% RSLogix 500 project LVD211007_994.RSS, saved by version 12.00.00.00 %
PROJECT "LINL0619"    % processor: MicroLogix 1400 %

PROGRAM FILES
  LAD 2 "MAIN"  70 rungs  % Main Program Routine %
  LAD 3 "FAST_TRIG"  9 rungs
  LAD 4 "ENABLES"  19 rungs
  LAD 5 "FEED"  14 rungs  % normal %
  LAD 6 "SPEEDS"  22 rungs
  LAD 7 "HSC BOT"  5 rungs
  LAD 8 "HSC TOP"  5 rungs
  LAD 9 "1 MS STI"  25 rungs  % high speed %
  LAD 10 "SHIFT BOT"  5 rungs
  LAD 11 "SHIFT TOP"  6 rungs
  LAD 12 "BOTOPTIC"  3 rungs
  LAD 13 "BOTOPTMES"  7 rungs
  LAD 14 "SHIFT TOP2"  7 rungs  % shift top inspection 6 %
  LAD 81 "I1"  25 rungs
  LAD 82 "I1 RESULT"  12 rungs
  LAD 83 "I1 PASS"  3 rungs
  LAD 84 "I1 FAIL"  3 rungs
  LAD 85 "I1 ACQ"  9 rungs
  LAD 86 "I1 TESTER"  5 rungs
  LAD 87 "I1 TRIG"  5 rungs
  LAD 88 "NO FIFO"  1 rungs
  LAD 89 "NO FIFO"  1 rungs
  LAD 90 "I1 DATA"  3 rungs
  LAD 91 "I1 FAULT"  9 rungs
  LAD 92 "I1 FIX1"  5 rungs
  LAD 93 "I1 FIX2"  3 rungs
  LAD 94 "I2"  24 rungs
  LAD 95 "I2 RESULT"  11 rungs
  LAD 96 "I2 PASS"  3 rungs
  LAD 97 "I2 FAIL"  3 rungs
  LAD 98 "I2 ACQ"  8 rungs
  LAD 99 "I2 TESTER"  9 rungs
  LAD 100 "I2 TRIG"  5 rungs
  LAD 101 "I2 FIFOSET"  7 rungs
  LAD 102 "I2 FIFOGET"  8 rungs
  LAD 103 "I2 DATA"  3 rungs
  LAD 104 "I2 FAULT"  9 rungs
  LAD 105 "I2 FIX1"  7 rungs
  LAD 106 "I2 FIX2"  3 rungs
  LAD 107 "I3"  1 rungs
  LAD 108 "I3 RESULT"  1 rungs
  LAD 109 "I3 PASS"  1 rungs
  LAD 110 "I3 FAIL"  1 rungs
  LAD 111 "I3 ACQ"  1 rungs
  LAD 112 "I3 TESTER"  1 rungs
  LAD 113 "I3 TRIG"  1 rungs
  LAD 114 "I3 FIFOSET"  1 rungs
  LAD 115 "I3 FIFOGET"  1 rungs
  LAD 116 "I3 DATA"  1 rungs
  LAD 117 "I3 FAULT"  1 rungs
  LAD 118 "I3 FIX1"  1 rungs
  LAD 119 "I3 FIX2"  1 rungs
  LAD 120 "I4"  1 rungs
  LAD 121 "I4 RESULT"  1 rungs
  LAD 122 "I4 PASS"  1 rungs
  LAD 123 "I4 FAIL"  1 rungs
  LAD 124 "I4 ACQ"  1 rungs
  LAD 125 "I4 TESTER"  1 rungs
  LAD 126 "I4 TRIG"  1 rungs
  LAD 127 "I4 FIFOSET"  1 rungs
  LAD 128 "I4 FIFOGET"  1 rungs
  LAD 129 "I4 DATA"  1 rungs
  LAD 130 "I4 FAULT"  1 rungs
  LAD 131 "I4 FIX1"  1 rungs
  LAD 132 "I4 FIX2"  1 rungs
  LAD 135 "XFER"  3 rungs
  LAD 137 "TOPOPTIC"  9 rungs
  LAD 138 "TOPOPVERT"  13 rungs
  LAD 139 "TOPOPREAL"  20 rungs
  LAD 140 "CT ALIGNS"  8 rungs
  LAD 142 "SET GOOD"  5 rungs
  LAD 148 "I5"  21 rungs
  LAD 149 "I5 RESULT"  7 rungs
  LAD 150 "I5 PASS"  6 rungs
  LAD 151 "I5 FAIL"  4 rungs
  LAD 152 "I5 ACQ"  9 rungs
  LAD 153 "I5 TESTER"  5 rungs
  LAD 154 "I5 TRIG"  5 rungs
  LAD 155 "I5 FIFOSET"  10 rungs
  LAD 156 "I5 FIFOGET"  8 rungs
  LAD 157 "I5 DATA"  3 rungs
  LAD 158 "I5 FAULT"  9 rungs
  LAD 159 "I5 FIX1"  5 rungs
  LAD 160 "I5 FIX2"  3 rungs
  LAD 161 "I6"  21 rungs
  LAD 162 "I6 RESULT"  7 rungs
  LAD 163 "I6 PASS"  5 rungs
  LAD 164 "I6 FAIL"  3 rungs
  LAD 165 "I6 ACQ"  8 rungs
  LAD 166 "I6 TESTER"  5 rungs
  LAD 167 "I6 TRIG"  5 rungs
  LAD 168 "I6 FIFOSET"  9 rungs
  LAD 169 "I6 FIFOGET"  8 rungs
  LAD 170 "I6 DATA"  3 rungs
  LAD 171 "I6 FAULT"  9 rungs
  LAD 172 "I6 FIX1"  5 rungs
  LAD 173 "I6 FIX2"  3 rungs
  LAD 174 "I7"  22 rungs
  LAD 175 "I7 RESULT"  13 rungs
  LAD 176 "I7 PASS"  3 rungs
  LAD 177 "I7 FAIL"  3 rungs
  LAD 178 "I7 ACQ"  9 rungs
  LAD 179 "I7 TESTER"  5 rungs
  LAD 180 "I7 TRIG"  5 rungs
  LAD 181 "I7 FIFOSET"  9 rungs
  LAD 182 "I7 FIFOGET"  8 rungs
  LAD 183 "I7 DATA"  3 rungs
  LAD 184 "I7 FAULT"  9 rungs
  LAD 185 "I7 FIX1"  5 rungs
  LAD 186 "I7 FIX2"  3 rungs
  LAD 187 "I8"  24 rungs
  LAD 188 "I8 RESULT"  13 rungs
  LAD 189 "I8 PASS"  3 rungs
  LAD 190 "I8 FAIL"  3 rungs
  LAD 191 "I8 ACQ"  9 rungs
  LAD 192 "I8 TESTER"  5 rungs
  LAD 193 "I8 TRIG"  5 rungs
  LAD 194 "I8 FIFOSET"  9 rungs
  LAD 195 "I8 FIFOGET"  8 rungs
  LAD 196 "I8 DATA"  3 rungs
  LAD 197 "I8 FAULT"  9 rungs
  LAD 198 "I8 FIX1"  5 rungs
  LAD 199 "I8 FIX2"  3 rungs
  LAD 200 "PASS BLOW"  18 rungs
  LAD 235 "TESTTRIGS"  7 rungs  % highspeed test triggers, not necessary %
  LAD 236 "TESTTRIG1"  5 rungs
  LAD 237 "TESTTRIG2"  4 rungs
  LAD 238 "TESTTRIG3"  4 rungs
  LAD 239 "TESTTRIG4"  4 rungs
  LAD 240 "TESTTRIG5"  4 rungs
  LAD 241 "TESTTRIG6"  4 rungs
  LAD 242 "TESTTRIG7"  4 rungs
  LAD 243 "TESTTRIG8"  4 rungs
  LAD 244 "PACKAGER"  31 rungs  % normal %
  LAD 245 "NO PACKAGE"  8 rungs
  LAD 246 "RATE1"  9 rungs
  LAD 247 "RATE2"  6 rungs
  LAD 248 "RESET RATE"  6 rungs
  LAD 249 "NP STOP"  8 rungs  % stop on no good %
  LAD 250 "SPEED BOT"  8 rungs  % high speed %
  LAD 251 "SPEED TOP"  8 rungs  % high speed %
  LAD 252 "P BOT"  7 rungs  % high speed %
  LAD 253 "P TOP"  7 rungs  % high speed %
  LAD 254 "TOTALCOUNT"  4 rungs
  LAD 255 "SAVED"  32 rungs
  LAD 141, 143, 144: only END

DATA FILES
  O0 OUTPUT  11 elements
  I1 INPUT  11 elements
  S2 STATUS  66 elements
  B3 BINARY  256 elements
  T4 TIMER  45 elements
  C5 COUNTER  1 elements
  R6 CONTROL  30 elements
  N7 INTEGER  200 elements
  F8 FLOAT  1 elements
  L13 LONG  256 elements
  L19 RATE DATA  50 elements
  L20 I7TIMEFIFO  256 elements
  L21 I7POSFIFO  256 elements
  L22 I8TIMEFIFO  50 elements
  L23 I8POSFIFO  50 elements
  L30 INS5TIME  50 elements
  L31 INS5POS  50 elements
  L32 INS6TIME  50 elements
  L33 INS6POS  50 elements
  B34 BOT NG  128 elements
  B35 TOP NG  128 elements
  B36 BOT OK  128 elements
  B37 TOP OK 1  128 elements
  B38 EX1 TEST  1 elements
  B39 TOP OK 2  128 elements
  B40 EX2 TEST  1 elements
  B41 TOP OK 3  128 elements
  B100 NEW HMI B  100 elements
  N101 NEW HMI N  256 elements
  L102 NEW HMI L  256 elements

LADDER 2 "MAIN"    % Main Program Routine %
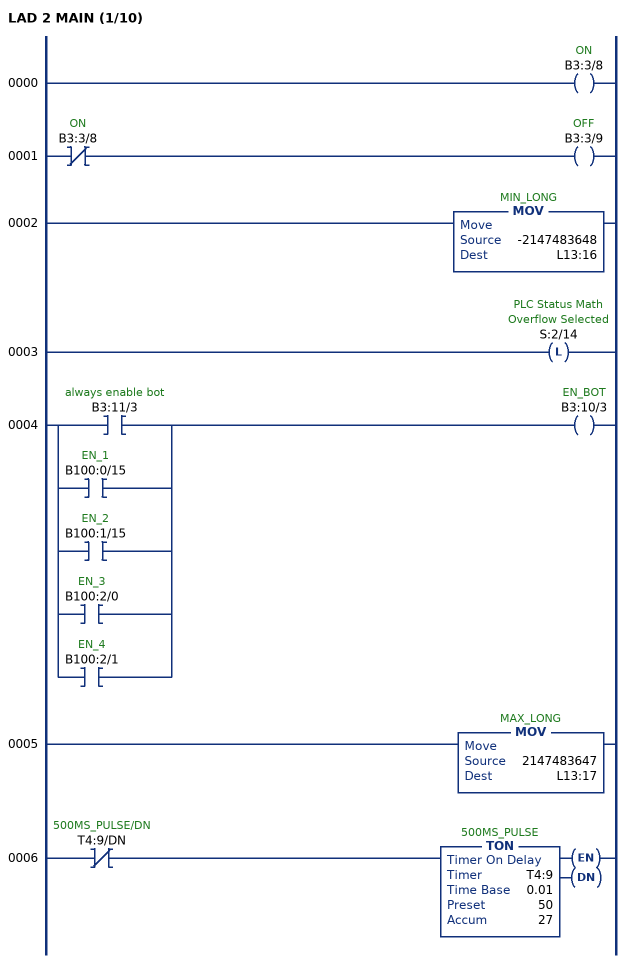
% Rung: 0 %
SOR OTE B3:3/8 EOR
%   B3:3/8  ON %
% Rung: 1 %
SOR XIO B3:3/8 OTE B3:3/9 EOR
%   B3:3/8  ON %
%   B3:3/9  OFF %
% Rung: 2 %
SOR MOV -2147483648 L13:16 EOR
%   L13:16  MIN_LONG %
% Rung: 3 %
SOR OTL S:2/14 EOR
%   S:2/14  "PLC Status Math Overflow Selected" %
% Rung: 4 %
SOR BST XIC B3:11/3 NXB XIC B100:0/15 NXB XIC B100:1/15 NXB XIC B100:2/0 NXB XIC B100:2/1 BND OTE B3:10/3 EOR
%   B3:11/3  "always enable bot" %
%   B100:0/15  EN_1 %
%   B100:1/15  EN_2 %
%   B100:2/0  EN_3 %
%   B100:2/1  EN_4 %
%   B3:10/3  EN_BOT %
% Rung: 5 %
SOR MOV 2147483647 L13:17 EOR
%   L13:17  MAX_LONG %
% Rung: 6 %
SOR XIO T4:9/DN TON T4:9 0.01 50 27 EOR
%   T4:9  500MS_PULSE %

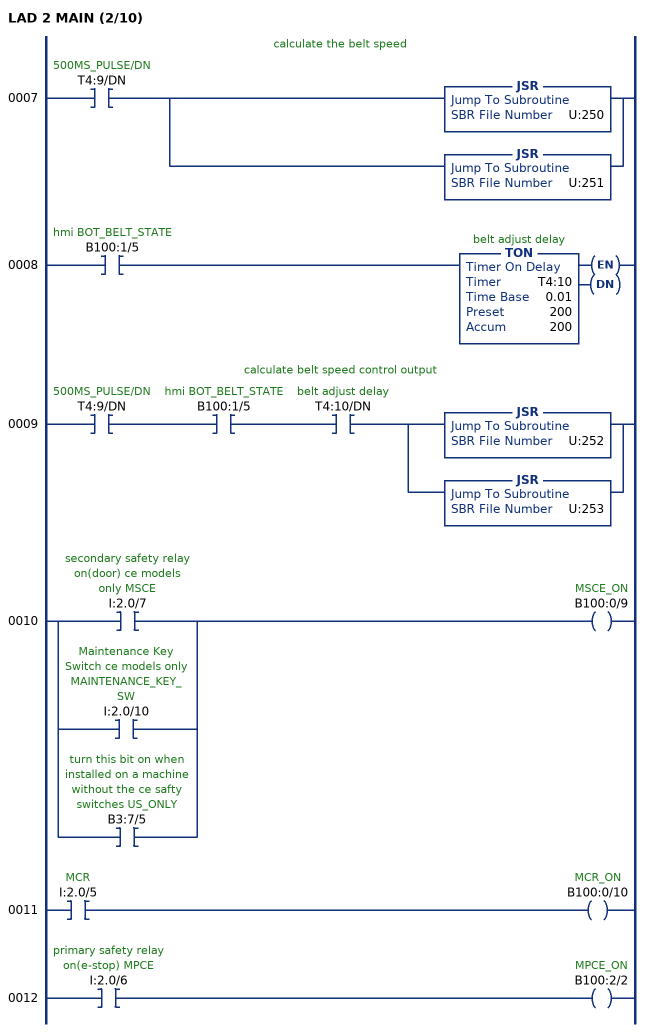
% Rung: 7 %
% calculate the belt speed %
SOR XIC T4:9/DN BST JSR U:250 NXB JSR U:251 BND EOR
%   T4:9  500MS_PULSE %
% Rung: 8 %
SOR XIC B100:1/5 TON T4:10 0.01 200 200 EOR
%   B100:1/5  BOT_BELT_STATE  "hmi" %
%   T4:10  "belt adjust delay" %
% Rung: 9 %
% calculate belt speed control output %
SOR XIC T4:9/DN XIC B100:1/5 XIC T4:10/DN BST JSR U:252 NXB JSR U:253 BND EOR
%   T4:9  500MS_PULSE %
%   B100:1/5  BOT_BELT_STATE  "hmi" %
%   T4:10  "belt adjust delay" %
% Rung: 10 %
SOR BST XIC I:2.0/7 NXB XIC I:2.0/10 NXB XIC B3:7/5 BND OTE B100:0/9 EOR
%   I:2.0/7  MSCE  "secondary safety relay on(door) ce models only" %
%   I:2.0/10  MAINTENANCE_KEY_SW  "Maintenance Key Switch ce models only" %
%   B3:7/5  US_ONLY  "turn this bit on when installed on a machine without the ce safty switches" %
%   B100:0/9  MSCE_ON %
% Rung: 11 %
SOR XIC I:2.0/5 OTE B100:0/10 EOR
%   I:2.0/5  MCR %
%   B100:0/10  MCR_ON %
% Rung: 12 %
SOR XIC I:2.0/6 OTE B100:2/2 EOR
%   I:2.0/6  MPCE  "primary safety relay on(e-stop)" %
%   B100:2/2  MPCE_ON %

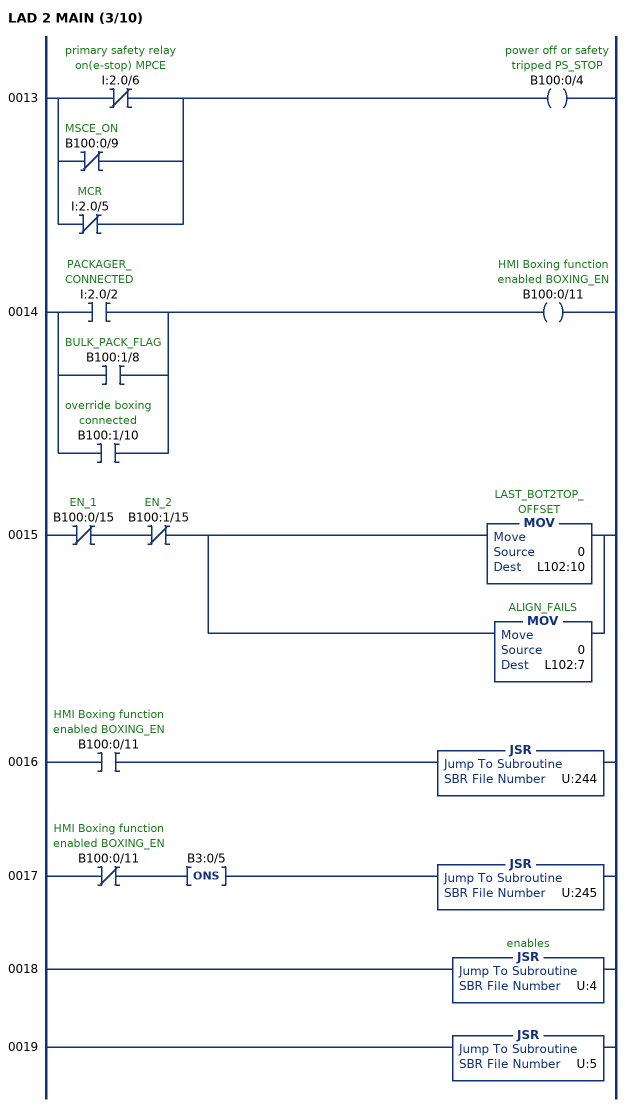
% Rung: 13 %
SOR BST XIO I:2.0/6 NXB XIO B100:0/9 NXB XIO I:2.0/5 BND OTE B100:0/4 EOR
%   I:2.0/6  MPCE  "primary safety relay on(e-stop)" %
%   B100:0/9  MSCE_ON %
%   I:2.0/5  MCR %
%   B100:0/4  PS_STOP  "power off or safety tripped" %
% Rung: 14 %
SOR BST XIC I:2.0/2 NXB XIC B100:1/8 NXB XIC B100:1/10 BND OTE B100:0/11 EOR
%   I:2.0/2  PACKAGER_CONNECTED %
%   B100:1/8  BULK_PACK_FLAG %
%   B100:1/10  "override boxing connected" %
%   B100:0/11  BOXING_EN  "HMI Boxing function enabled" %
% Rung: 15 %
SOR XIO B100:0/15 XIO B100:1/15 BST MOV 0 L102:10 NXB MOV 0 L102:7 BND EOR
%   B100:0/15  EN_1 %
%   B100:1/15  EN_2 %
%   L102:10  LAST_BOT2TOP_OFFSET %
%   L102:7  ALIGN_FAILS %
% Rung: 16 %
SOR XIC B100:0/11 JSR U:244 EOR
%   B100:0/11  BOXING_EN  "HMI Boxing function enabled" %
% Rung: 17 %
SOR XIO B100:0/11 ONS B3:0/5 JSR U:245 EOR
%   B100:0/11  BOXING_EN  "HMI Boxing function enabled" %
% Rung: 18 %
SOR JSR U:4 EOR
%   U:4  "enables" %
% Rung: 19 %
SOR JSR U:5 EOR

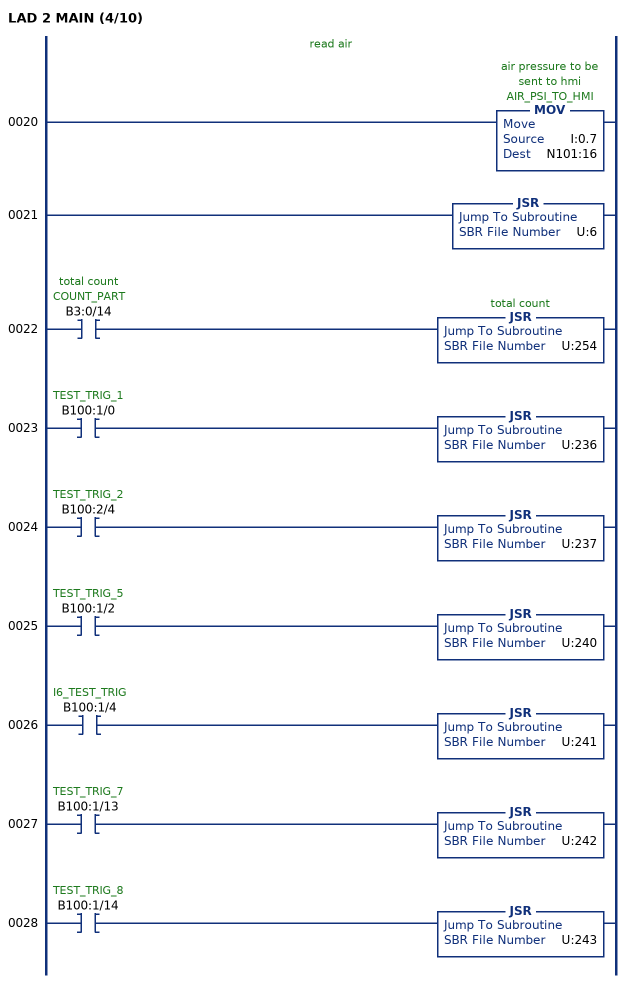
% Rung: 20 %
% read air %
SOR MOV I:0.7 N101:16 EOR
%   I:0.7  "Air Presure Sensor Input Signal" %
%   N101:16  AIR_PSI_TO_HMI  "air pressure to be sent to hmi" %
% Rung: 21 %
SOR JSR U:6 EOR
% Rung: 22 %
SOR XIC B3:0/14 JSR U:254 EOR
%   B3:0/14  COUNT_PART  "total count" %
%   U:254  "total count" %
% Rung: 23 %
SOR XIC B100:1/0 JSR U:236 EOR
%   B100:1/0  TEST_TRIG_1 %
% Rung: 24 %
SOR XIC B100:2/4 JSR U:237 EOR
%   B100:2/4  TEST_TRIG_2 %
% Rung: 25 %
SOR XIC B100:1/2 JSR U:240 EOR
%   B100:1/2  TEST_TRIG_5 %
% Rung: 26 %
SOR XIC B100:1/4 JSR U:241 EOR
%   B100:1/4  I6_TEST_TRIG %
% Rung: 27 %
SOR XIC B100:1/13 JSR U:242 EOR
%   B100:1/13  TEST_TRIG_7 %
% Rung: 28 %
SOR XIC B100:1/14 JSR U:243 EOR
%   B100:1/14  TEST_TRIG_8 %

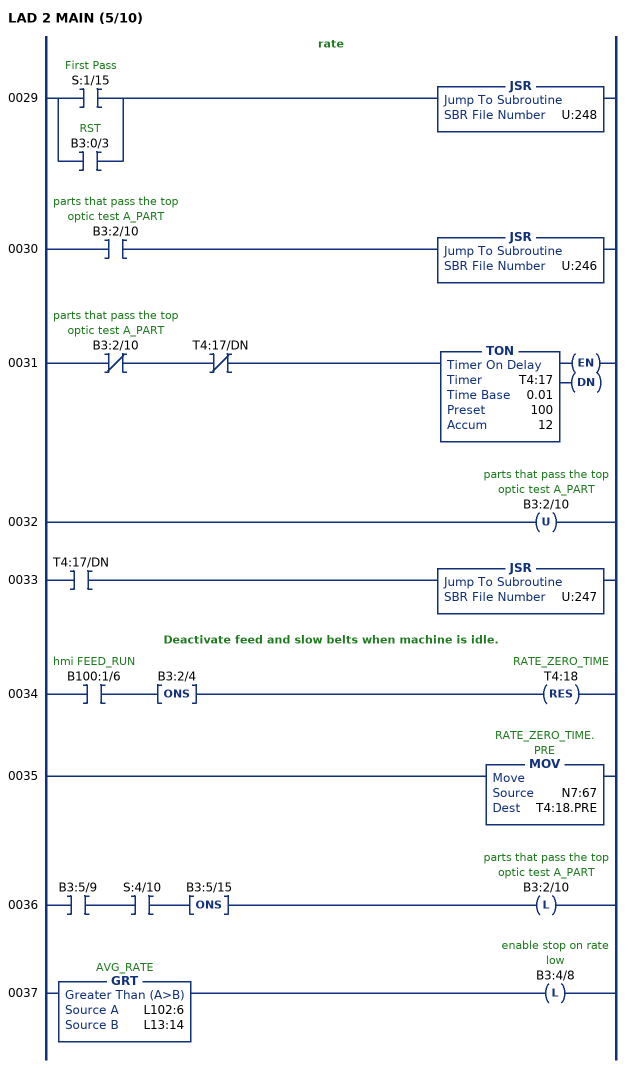
% Rung: 29 %
% TITLE: rate %
SOR BST XIC S:1/15 NXB XIC B3:0/3 BND JSR U:248 EOR
%   S:1/15  "First Pass" %
%   B3:0/3  RST %
% Rung: 30 %
SOR XIC B3:2/10 JSR U:246 EOR
%   B3:2/10  A_PART  "parts that pass the top optic test" %
% Rung: 31 %
SOR XIO B3:2/10 XIO T4:17/DN TON T4:17 0.01 100 12 EOR
%   B3:2/10  A_PART  "parts that pass the top optic test" %
% Rung: 32 %
SOR OTU B3:2/10 EOR
%   B3:2/10  A_PART  "parts that pass the top optic test" %
% Rung: 33 %
SOR XIC T4:17/DN JSR U:247 EOR
% Rung: 34 %
% TITLE: Deactivate feed and slow belts when machine is idle. %
SOR XIC B100:1/6 ONS B3:2/4 RES T4:18 EOR
%   B100:1/6  FEED_RUN  "hmi" %
%   T4:18  RATE_ZERO_TIME %
% Rung: 35 %
SOR MOV N7:67 T4:18.PRE EOR
%   N7:67  "empty bowl or jam bowl run time" %
%   T4:18  RATE_ZERO_TIME %
% Rung: 36 %
SOR XIC B3:5/9 XIC S:4/10 ONS B3:5/15 OTL B3:2/10 EOR
%   B3:2/10  A_PART  "parts that pass the top optic test" %
% Rung: 37 %
SOR GRT L102:6 L13:14 OTL B3:4/8 EOR
%   L102:6  AVG_RATE %
%   B3:4/8  "enable stop on rate low" %

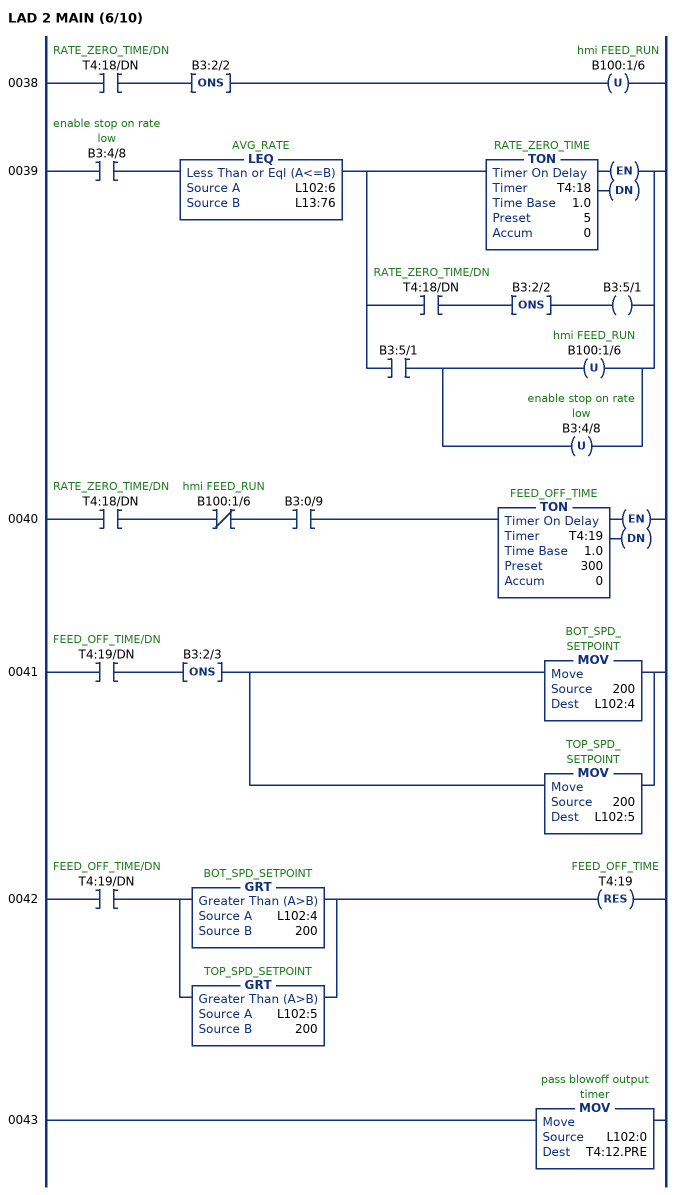
% Rung: 38 %
SOR XIC T4:18/DN ONS B3:2/2 OTU B100:1/6 EOR
%   T4:18  RATE_ZERO_TIME %
%   B100:1/6  FEED_RUN  "hmi" %
% Rung: 39 %
SOR XIC B3:4/8 LEQ L102:6 L13:76 BST TON T4:18 1.0 5 0 NXB XIC T4:18/DN ONS B3:2/2 OTE B3:5/1 NXB XIC B3:5/1 BST OTU B100:1/6 NXB OTU B3:4/8 BND BND EOR
%   B3:4/8  "enable stop on rate low" %
%   L102:6  AVG_RATE %
%   T4:18  RATE_ZERO_TIME %
%   B100:1/6  FEED_RUN  "hmi" %
% Rung: 40 %
SOR XIC T4:18/DN XIO B100:1/6 XIC B3:0/9 TON T4:19 1.0 300 0 EOR
%   T4:18  RATE_ZERO_TIME %
%   B100:1/6  FEED_RUN  "hmi" %
%   T4:19  FEED_OFF_TIME %
% Rung: 41 %
SOR XIC T4:19/DN ONS B3:2/3 BST MOV 200 L102:4 NXB MOV 200 L102:5 BND EOR
%   T4:19  FEED_OFF_TIME %
%   L102:4  BOT_SPD_SETPOINT %
%   L102:5  TOP_SPD_SETPOINT %
% Rung: 42 %
SOR XIC T4:19/DN BST GRT L102:4 200 NXB GRT L102:5 200 BND RES T4:19 EOR
%   T4:19  FEED_OFF_TIME %
%   L102:4  BOT_SPD_SETPOINT %
%   L102:5  TOP_SPD_SETPOINT %
% Rung: 43 %
SOR MOV L102:0 T4:12.PRE EOR
%   L102:0  BLOW_TIME %
%   T4:12  "pass blowoff output timer" %

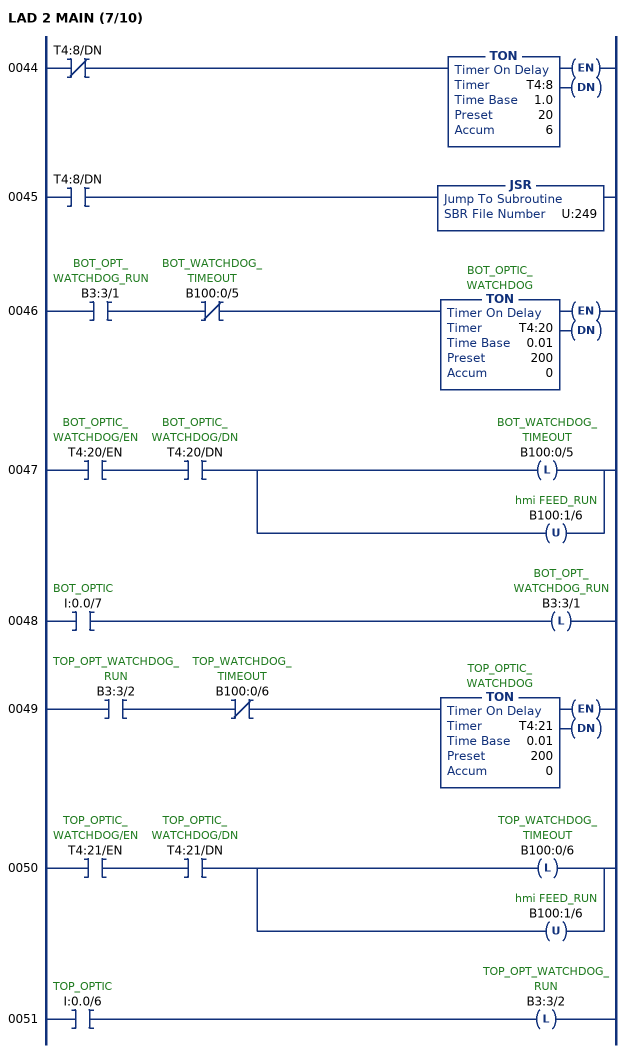
% Rung: 44 %
SOR XIO T4:8/DN TON T4:8 1.0 20 6 EOR
% Rung: 45 %
SOR XIC T4:8/DN JSR U:249 EOR
% Rung: 46 %
SOR XIC B3:3/1 XIO B100:0/5 TON T4:20 0.01 200 0 EOR
%   B3:3/1  BOT_OPT_WATCHDOG_RUN %
%   B100:0/5  BOT_WATCHDOG_TIMEOUT %
%   T4:20  BOT_OPTIC_WATCHDOG %
% Rung: 47 %
SOR XIC T4:20/EN XIC T4:20/DN BST OTL B100:0/5 NXB OTU B100:1/6 BND EOR
%   T4:20  BOT_OPTIC_WATCHDOG %
%   B100:0/5  BOT_WATCHDOG_TIMEOUT %
%   B100:1/6  FEED_RUN  "hmi" %
% Rung: 48 %
SOR XIC I:0.0/7 OTL B3:3/1 EOR
%   I:0.0/7  BOT_OPTIC %
%   B3:3/1  BOT_OPT_WATCHDOG_RUN %
% Rung: 49 %
SOR XIC B3:3/2 XIO B100:0/6 TON T4:21 0.01 200 0 EOR
%   B3:3/2  TOP_OPT_WATCHDOG_RUN %
%   B100:0/6  TOP_WATCHDOG_TIMEOUT %
%   T4:21  TOP_OPTIC_WATCHDOG %
% Rung: 50 %
SOR XIC T4:21/EN XIC T4:21/DN BST OTL B100:0/6 NXB OTU B100:1/6 BND EOR
%   T4:21  TOP_OPTIC_WATCHDOG %
%   B100:0/6  TOP_WATCHDOG_TIMEOUT %
%   B100:1/6  FEED_RUN  "hmi" %
% Rung: 51 %
SOR XIC I:0.0/6 OTL B3:3/2 EOR
%   I:0.0/6  TOP_OPTIC %
%   B3:3/2  TOP_OPT_WATCHDOG_RUN %

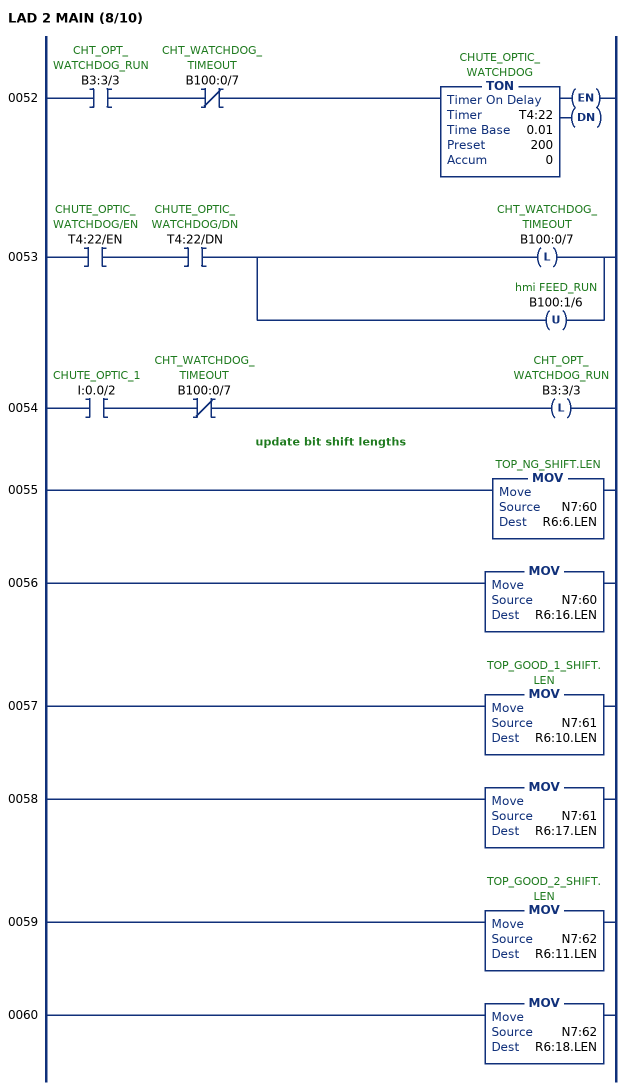
% Rung: 52 %
SOR XIC B3:3/3 XIO B100:0/7 TON T4:22 0.01 200 0 EOR
%   B3:3/3  CHT_OPT_WATCHDOG_RUN %
%   B100:0/7  CHT_WATCHDOG_TIMEOUT %
%   T4:22  CHUTE_OPTIC_WATCHDOG %
% Rung: 53 %
SOR XIC T4:22/EN XIC T4:22/DN BST OTL B100:0/7 NXB OTU B100:1/6 BND EOR
%   T4:22  CHUTE_OPTIC_WATCHDOG %
%   B100:0/7  CHT_WATCHDOG_TIMEOUT %
%   B100:1/6  FEED_RUN  "hmi" %
% Rung: 54 %
SOR XIC I:0.0/2 XIO B100:0/7 OTL B3:3/3 EOR
%   I:0.0/2  CHUTE_OPTIC_1 %
%   B100:0/7  CHT_WATCHDOG_TIMEOUT %
%   B3:3/3  CHT_OPT_WATCHDOG_RUN %
% Rung: 55 %
% TITLE: update bit shift lengths %
SOR MOV N7:60 R6:6.LEN EOR
%   R6:6  TOP_NG_SHIFT %
% Rung: 56 %
SOR MOV N7:60 R6:16.LEN EOR
% Rung: 57 %
SOR MOV N7:61 R6:10.LEN EOR
%   R6:10  TOP_GOOD_1_SHIFT %
% Rung: 58 %
SOR MOV N7:61 R6:17.LEN EOR
% Rung: 59 %
SOR MOV N7:62 R6:11.LEN EOR
%   R6:11  TOP_GOOD_2_SHIFT %
% Rung: 60 %
SOR MOV N7:62 R6:18.LEN EOR

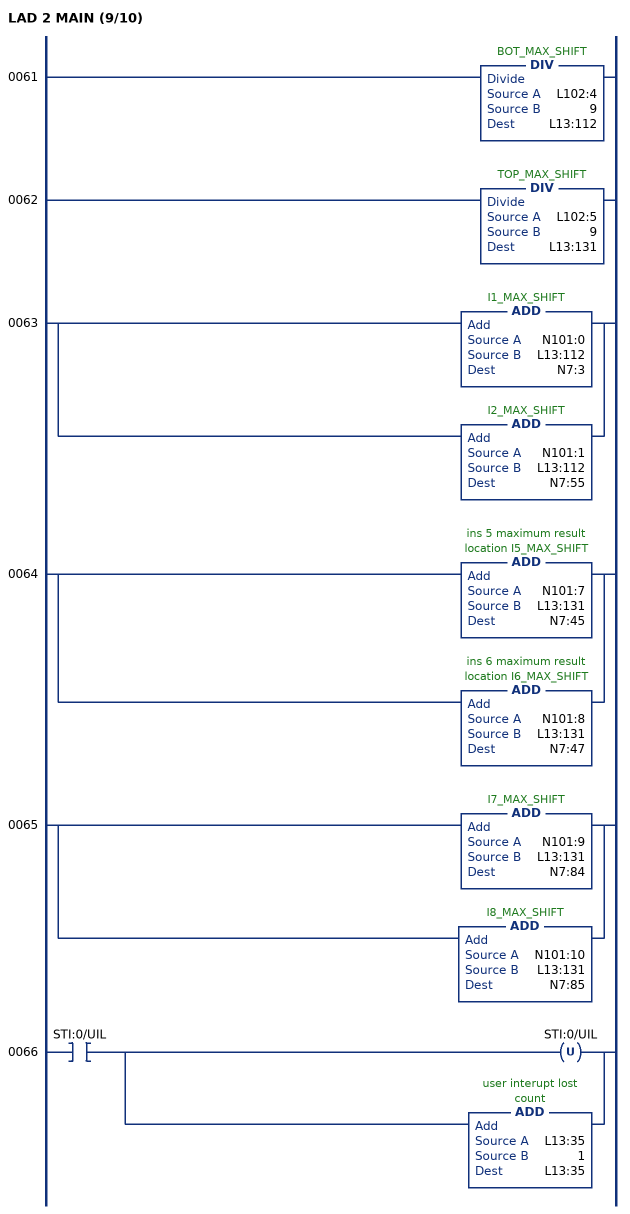
% Rung: 61 %
SOR DIV L102:4 9 L13:112 EOR
%   L102:4  BOT_SPD_SETPOINT %
%   L13:112  BOT_MAX_SHIFT %
% Rung: 62 %
SOR DIV L102:5 9 L13:131 EOR
%   L102:5  TOP_SPD_SETPOINT %
%   L13:131  TOP_MAX_SHIFT %
% Rung: 63 %
SOR BST ADD N101:0 L13:112 N7:3 NXB ADD N101:1 L13:112 N7:55 BND EOR
%   N101:0  I1_TRIG_LOC %
%   L13:112  BOT_MAX_SHIFT %
%   N7:3  I1_MAX_SHIFT %
%   N101:1  I2_TRIG_LOC %
%   N7:55  I2_MAX_SHIFT %
% Rung: 64 %
SOR BST ADD N101:7 L13:131 N7:45 NXB ADD N101:8 L13:131 N7:47 BND EOR
%   N101:7  I5_TRIG_LOC %
%   L13:131  TOP_MAX_SHIFT %
%   N7:45  I5_MAX_SHIFT  "ins 5 maximum result location" %
%   N101:8  I6_TRIG_LOC %
%   N7:47  I6_MAX_SHIFT  "ins 6 maximum result location" %
% Rung: 65 %
SOR BST ADD N101:9 L13:131 N7:84 NXB ADD N101:10 L13:131 N7:85 BND EOR
%   N101:9  I7_TRIG_LOC %
%   L13:131  TOP_MAX_SHIFT %
%   N7:84  I7_MAX_SHIFT %
%   N101:10  I8_TRIG_LOC %
%   N7:85  I8_MAX_SHIFT %
% Rung: 66 %
SOR XIC STI:0/UIL BST OTU STI:0/UIL NXB ADD L13:35 1 L13:35 BND EOR
%   L13:35  "user interupt lost count" %

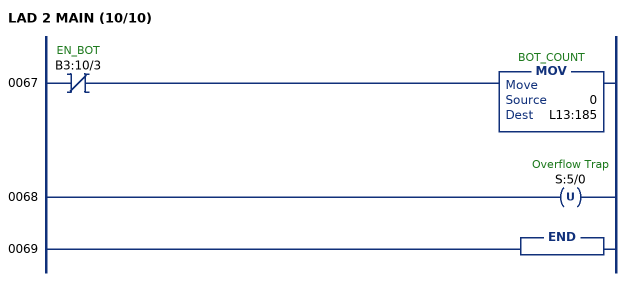
% Rung: 67 %
SOR XIO B3:10/3 MOV 0 L13:185 EOR
%   B3:10/3  EN_BOT %
%   L13:185  BOT_COUNT %
% Rung: 68 %
SOR OTU S:5/0 EOR
%   S:5/0  "Overflow Trap" %
% Rung: 69 %
SOR END EOR

LADDER 3 "FAST_TRIG"
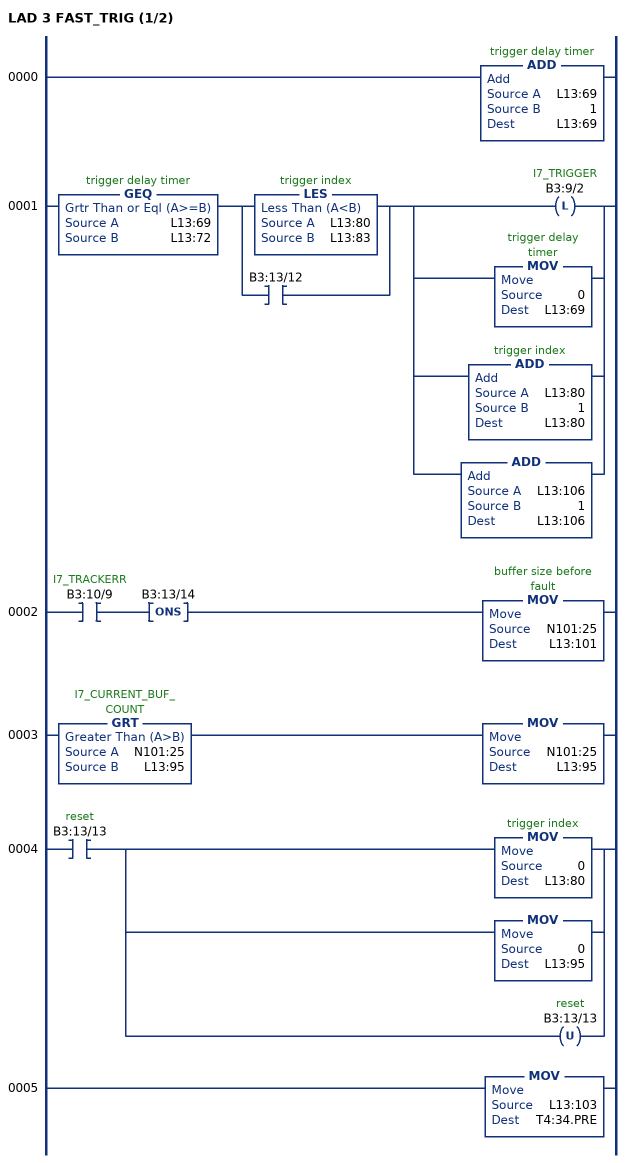
% Rung: 0 %
SOR ADD L13:69 1 L13:69 EOR
%   L13:69  "trigger delay timer" %
% Rung: 1 %
SOR GEQ L13:69 L13:72 BST LES L13:80 L13:83 NXB XIC B3:13/12 BND BST OTL B3:9/2 NXB MOV 0 L13:69 NXB ADD L13:80 1 L13:80 NXB ADD L13:106 1 L13:106 BND EOR
%   L13:69  "trigger delay timer" %
%   L13:72  "time between triggers" %
%   L13:80  "trigger index" %
%   L13:83  "max triggers" %
%   B3:9/2  I7_TRIGGER %
% Rung: 2 %
SOR XIC B3:10/9 ONS B3:13/14 MOV N101:25 L13:101 EOR
%   B3:10/9  I7_TRACKERR %
%   N101:25  I7_CURRENT_BUF_COUNT %
%   L13:101  "buffer size before fault" %
% Rung: 3 %
SOR GRT N101:25 L13:95 MOV N101:25 L13:95 EOR
%   N101:25  I7_CURRENT_BUF_COUNT %
% Rung: 4 %
SOR XIC B3:13/13 BST MOV 0 L13:80 NXB MOV 0 L13:95 NXB OTU B3:13/13 BND EOR
%   B3:13/13  "reset" %
%   L13:80  "trigger index" %
% Rung: 5 %
SOR MOV L13:103 T4:34.PRE EOR

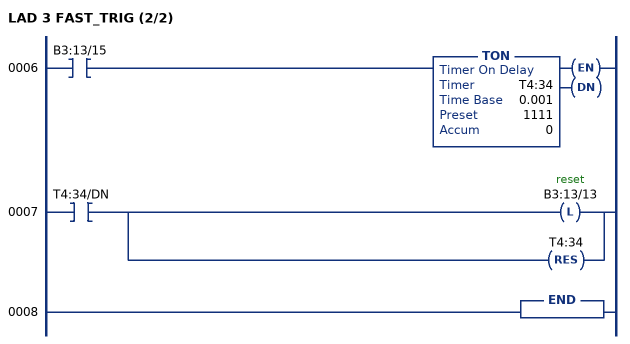
% Rung: 6 %
SOR XIC B3:13/15 TON T4:34 0.001 1111 0 EOR
% Rung: 7 %
SOR XIC T4:34/DN BST OTL B3:13/13 NXB RES T4:34 BND EOR
%   B3:13/13  "reset" %
% Rung: 8 %
SOR END EOR

LADDER 4 "ENABLES"
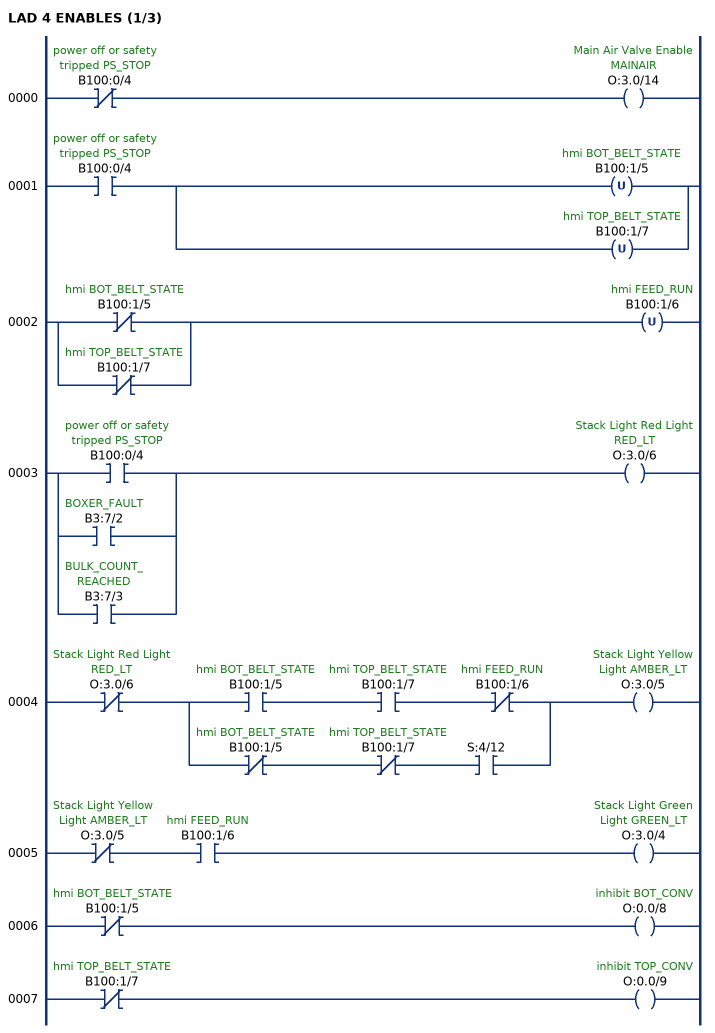
% Rung: 0 %
SOR XIO B100:0/4 OTE O:3.0/14 EOR
%   B100:0/4  PS_STOP  "power off or safety tripped" %
%   O:3.0/14  MAINAIR  "Main Air Valve Enable" %
% Rung: 1 %
SOR XIC B100:0/4 BST OTU B100:1/5 NXB OTU B100:1/7 BND EOR
%   B100:0/4  PS_STOP  "power off or safety tripped" %
%   B100:1/5  BOT_BELT_STATE  "hmi" %
%   B100:1/7  TOP_BELT_STATE  "hmi" %
% Rung: 2 %
SOR BST XIO B100:1/5 NXB XIO B100:1/7 BND OTU B100:1/6 EOR
%   B100:1/5  BOT_BELT_STATE  "hmi" %
%   B100:1/7  TOP_BELT_STATE  "hmi" %
%   B100:1/6  FEED_RUN  "hmi" %
% Rung: 3 %
SOR BST XIC B100:0/4 NXB XIC B3:7/2 NXB XIC B3:7/3 BND OTE O:3.0/6 EOR
%   B100:0/4  PS_STOP  "power off or safety tripped" %
%   B3:7/2  BOXER_FAULT %
%   B3:7/3  BULK_COUNT_REACHED %
%   O:3.0/6  RED_LT  "Stack Light Red Light" %
% Rung: 4 %
SOR XIO O:3.0/6 BST XIC B100:1/5 XIC B100:1/7 XIO B100:1/6 NXB XIO B100:1/5 XIO B100:1/7 XIC S:4/12 BND OTE O:3.0/5 EOR
%   O:3.0/6  RED_LT  "Stack Light Red Light" %
%   B100:1/5  BOT_BELT_STATE  "hmi" %
%   B100:1/7  TOP_BELT_STATE  "hmi" %
%   B100:1/6  FEED_RUN  "hmi" %
%   O:3.0/5  AMBER_LT  "Stack Light Yellow Light" %
% Rung: 5 %
SOR XIO O:3.0/5 XIC B100:1/6 OTE O:3.0/4 EOR
%   O:3.0/5  AMBER_LT  "Stack Light Yellow Light" %
%   B100:1/6  FEED_RUN  "hmi" %
%   O:3.0/4  GREEN_LT  "Stack Light Green Light" %
% Rung: 6 %
SOR XIO B100:1/5 OTE O:0.0/8 EOR
%   B100:1/5  BOT_BELT_STATE  "hmi" %
%   O:0.0/8  BOT_CONV  "inhibit" %
% Rung: 7 %
SOR XIO B100:1/7 OTE O:0.0/9 EOR
%   B100:1/7  TOP_BELT_STATE  "hmi" %
%   O:0.0/9  TOP_CONV  "inhibit" %

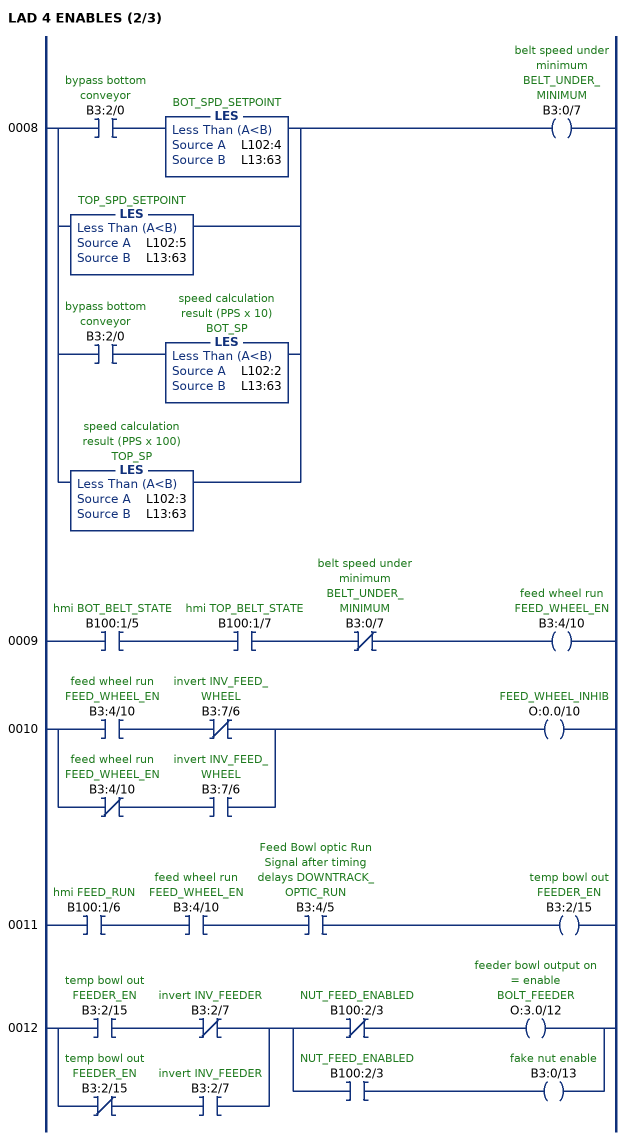
% Rung: 8 %
SOR BST XIC B3:2/0 LES L102:4 L13:63 NXB LES L102:5 L13:63 NXB XIC B3:2/0 LES L102:2 L13:63 NXB LES L102:3 L13:63 BND OTE B3:0/7 EOR
%   B3:2/0  "bypass bottom conveyor" %
%   L102:4  BOT_SPD_SETPOINT %
%   L13:63  "min belt speed" %
%   L102:5  TOP_SPD_SETPOINT %
%   L102:2  BOT_SP  "speed calculation result (PPS x 10)" %
%   L102:3  TOP_SP  "speed calculation result (PPS x 100)" %
%   B3:0/7  BELT_UNDER_MINIMUM  "belt speed under minimum" %
% Rung: 9 %
SOR XIC B100:1/5 XIC B100:1/7 XIO B3:0/7 OTE B3:4/10 EOR
%   B100:1/5  BOT_BELT_STATE  "hmi" %
%   B100:1/7  TOP_BELT_STATE  "hmi" %
%   B3:0/7  BELT_UNDER_MINIMUM  "belt speed under minimum" %
%   B3:4/10  FEED_WHEEL_EN  "feed wheel run" %
% Rung: 10 %
SOR BST XIC B3:4/10 XIO B3:7/6 NXB XIO B3:4/10 XIC B3:7/6 BND OTE O:0.0/10 EOR
%   B3:4/10  FEED_WHEEL_EN  "feed wheel run" %
%   B3:7/6  INV_FEED_WHEEL  "invert" %
%   O:0.0/10  FEED_WHEEL_INHIB %
% Rung: 11 %
SOR XIC B100:1/6 XIC B3:4/10 XIC B3:4/5 OTE B3:2/15 EOR
%   B100:1/6  FEED_RUN  "hmi" %
%   B3:4/10  FEED_WHEEL_EN  "feed wheel run" %
%   B3:4/5  DOWNTRACK_OPTIC_RUN  "Feed Bowl optic Run Signal after timing delays" %
%   B3:2/15  FEEDER_EN  "temp bowl out" %
% Rung: 12 %
SOR BST XIC B3:2/15 XIO B3:2/7 NXB XIO B3:2/15 XIC B3:2/7 BND BST XIO B100:2/3 OTE O:3.0/12 NXB XIC B100:2/3 OTE B3:0/13 BND EOR
%   B3:2/15  FEEDER_EN  "temp bowl out" %
%   B3:2/7  INV_FEEDER  "invert" %
%   B100:2/3  NUT_FEED_ENABLED %
%   O:3.0/12  BOLT_FEEDER  "feeder bowl output on = enable" %
%   B3:0/13  "fake nut enable" %

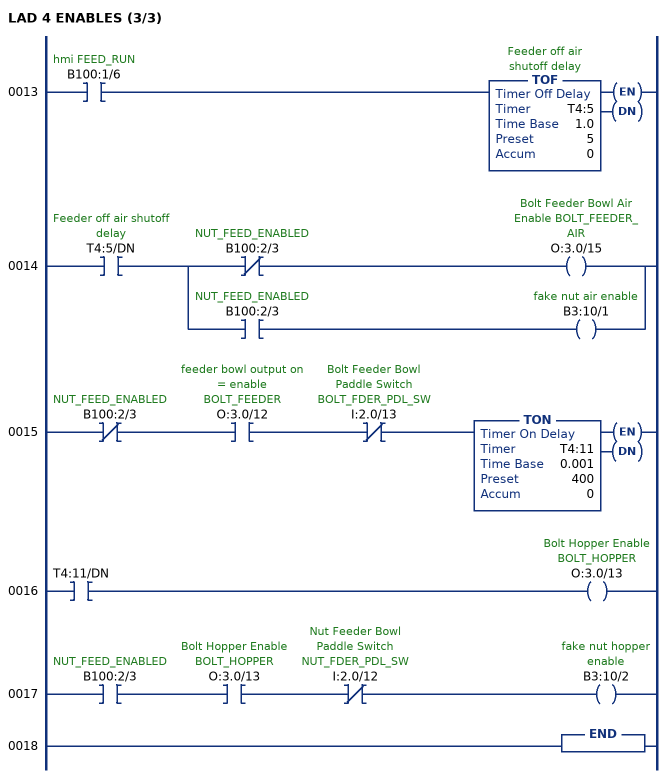
% Rung: 13 %
SOR XIC B100:1/6 TOF T4:5 1.0 5 0 EOR
%   B100:1/6  FEED_RUN  "hmi" %
%   T4:5  "Feeder off air shutoff delay" %
% Rung: 14 %
SOR XIC T4:5/DN BST XIO B100:2/3 OTE O:3.0/15 NXB XIC B100:2/3 OTE B3:10/1 BND EOR
%   T4:5  "Feeder off air shutoff delay" %
%   B100:2/3  NUT_FEED_ENABLED %
%   O:3.0/15  BOLT_FEEDER_AIR  "Bolt Feeder Bowl Air Enable" %
%   B3:10/1  "fake nut air enable" %
% Rung: 15 %
SOR XIO B100:2/3 XIC O:3.0/12 XIO I:2.0/13 TON T4:11 0.001 400 0 EOR
%   B100:2/3  NUT_FEED_ENABLED %
%   O:3.0/12  BOLT_FEEDER  "feeder bowl output on = enable" %
%   I:2.0/13  BOLT_FDER_PDL_SW  "Bolt Feeder Bowl Paddle Switch" %
% Rung: 16 %
SOR XIC T4:11/DN OTE O:3.0/13 EOR
%   O:3.0/13  BOLT_HOPPER  "Bolt Hopper Enable" %
% Rung: 17 %
SOR XIC B100:2/3 XIC O:3.0/13 XIO I:2.0/12 OTE B3:10/2 EOR
%   B100:2/3  NUT_FEED_ENABLED %
%   O:3.0/13  BOLT_HOPPER  "Bolt Hopper Enable" %
%   I:2.0/12  NUT_FDER_PDL_SW  "Nut Feeder Bowl Paddle Switch" %
%   B3:10/2  "fake nut hopper enable" %
% Rung: 18 %
SOR END EOR

LADDER 5 "FEED"    % normal %
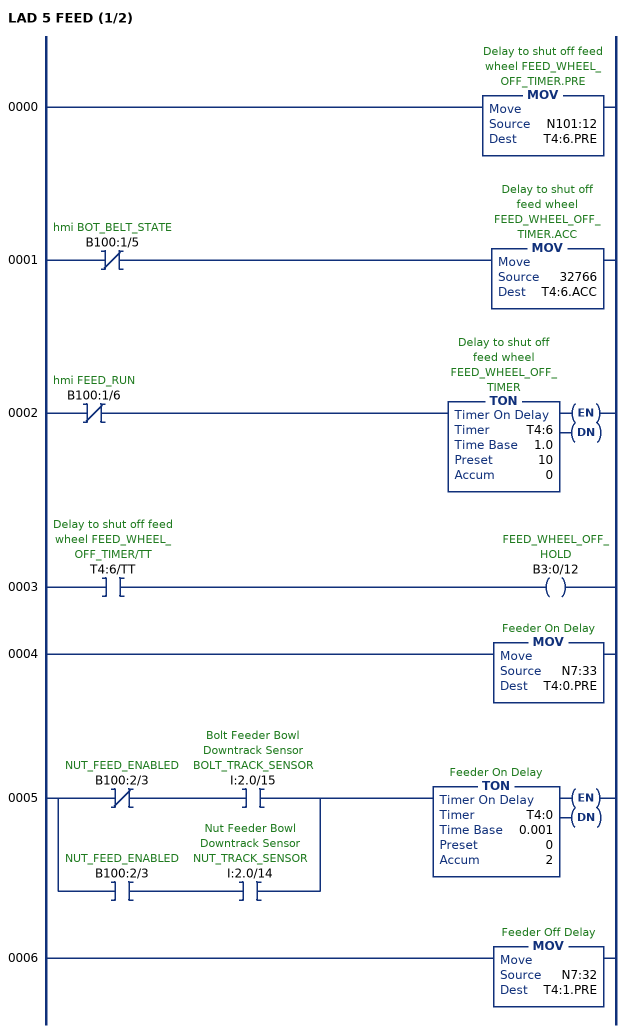
% Rung: 0 %
SOR MOV N101:12 T4:6.PRE EOR
%   N101:12  FEED_WHEEL_STOP_TIME %
%   T4:6  FEED_WHEEL_OFF_TIMER  "Delay to shut off feed wheel" %
% Rung: 1 %
SOR XIO B100:1/5 MOV 32766 T4:6.ACC EOR
%   B100:1/5  BOT_BELT_STATE  "hmi" %
%   T4:6  FEED_WHEEL_OFF_TIMER  "Delay to shut off feed wheel" %
% Rung: 2 %
SOR XIO B100:1/6 TON T4:6 1.0 10 0 EOR
%   B100:1/6  FEED_RUN  "hmi" %
%   T4:6  FEED_WHEEL_OFF_TIMER  "Delay to shut off feed wheel" %
% Rung: 3 %
SOR XIC T4:6/TT OTE B3:0/12 EOR
%   T4:6  FEED_WHEEL_OFF_TIMER  "Delay to shut off feed wheel" %
%   B3:0/12  FEED_WHEEL_OFF_HOLD %
% Rung: 4 %
SOR MOV N7:33 T4:0.PRE EOR
%   N7:33  "down track on delay" %
%   T4:0  "Feeder On Delay" %
% Rung: 5 %
SOR BST XIO B100:2/3 XIC I:2.0/15 NXB XIC B100:2/3 XIC I:2.0/14 BND TON T4:0 0.001 0 2 EOR
%   B100:2/3  NUT_FEED_ENABLED %
%   I:2.0/15  BOLT_TRACK_SENSOR  "Bolt Feeder Bowl Downtrack Sensor" %
%   I:2.0/14  NUT_TRACK_SENSOR  "Nut Feeder Bowl Downtrack Sensor" %
%   T4:0  "Feeder On Delay" %
% Rung: 6 %
SOR MOV N7:32 T4:1.PRE EOR
%   N7:32  "down track off delay" %
%   T4:1  "Feeder Off Delay" %

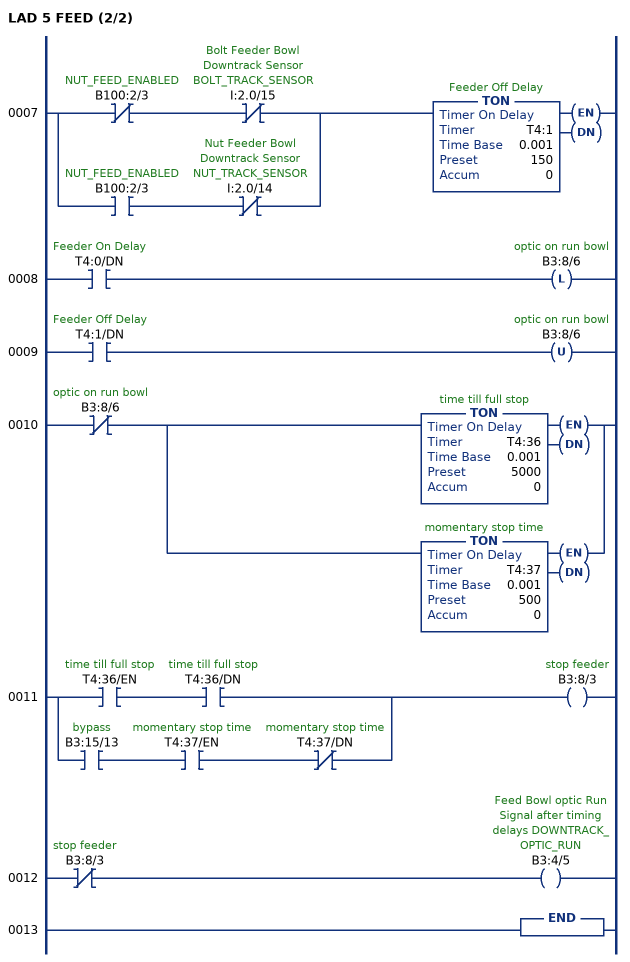
% Rung: 7 %
SOR BST XIO B100:2/3 XIO I:2.0/15 NXB XIC B100:2/3 XIO I:2.0/14 BND TON T4:1 0.001 150 0 EOR
%   B100:2/3  NUT_FEED_ENABLED %
%   I:2.0/15  BOLT_TRACK_SENSOR  "Bolt Feeder Bowl Downtrack Sensor" %
%   I:2.0/14  NUT_TRACK_SENSOR  "Nut Feeder Bowl Downtrack Sensor" %
%   T4:1  "Feeder Off Delay" %
% Rung: 8 %
SOR XIC T4:0/DN OTL B3:8/6 EOR
%   T4:0  "Feeder On Delay" %
%   B3:8/6  "optic on run bowl" %
% Rung: 9 %
SOR XIC T4:1/DN OTU B3:8/6 EOR
%   T4:1  "Feeder Off Delay" %
%   B3:8/6  "optic on run bowl" %
% Rung: 10 %
SOR XIO B3:8/6 BST TON T4:36 0.001 5000 0 NXB TON T4:37 0.001 500 0 BND EOR
%   B3:8/6  "optic on run bowl" %
%   T4:36  "time till full stop" %
%   T4:37  "momentary stop time" %
% Rung: 11 %
SOR BST XIC T4:36/EN XIC T4:36/DN NXB XIC B3:15/13 XIC T4:37/EN XIO T4:37/DN BND OTE B3:8/3 EOR
%   T4:36  "time till full stop" %
%   B3:15/13  "bypass" %
%   T4:37  "momentary stop time" %
%   B3:8/3  "stop feeder" %
% Rung: 12 %
SOR XIO B3:8/3 OTE B3:4/5 EOR
%   B3:8/3  "stop feeder" %
%   B3:4/5  DOWNTRACK_OPTIC_RUN  "Feed Bowl optic Run Signal after timing delays" %
% Rung: 13 %
SOR END EOR

LADDER 6 "SPEEDS"
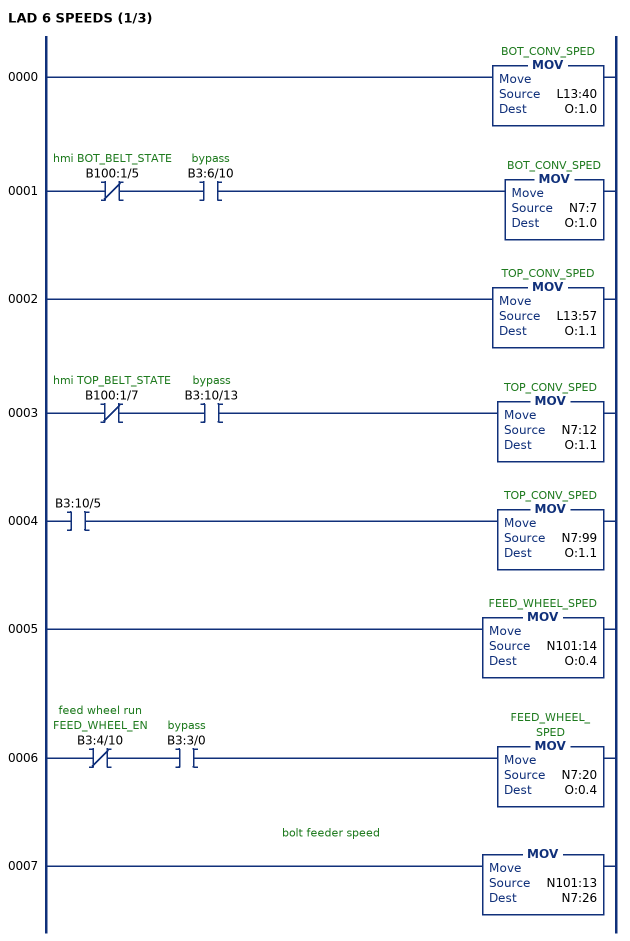
% Rung: 0 %
SOR MOV L13:40 O:1.0 EOR
%   L13:40  SCALED_BOT_VALUE %
%   O:1.0  BOT_CONV_SPED %
% Rung: 1 %
SOR XIO B100:1/5 XIC B3:6/10 MOV N7:7 O:1.0 EOR
%   B100:1/5  BOT_BELT_STATE  "hmi" %
%   B3:6/10  "bypass" %
%   O:1.0  BOT_CONV_SPED %
% Rung: 2 %
SOR MOV L13:57 O:1.1 EOR
%   L13:57  SCALED_TOP_VALUE %
%   O:1.1  TOP_CONV_SPED %
% Rung: 3 %
SOR XIO B100:1/7 XIC B3:10/13 MOV N7:12 O:1.1 EOR
%   B100:1/7  TOP_BELT_STATE  "hmi" %
%   B3:10/13  "bypass" %
%   O:1.1  TOP_CONV_SPED %
% Rung: 4 %
SOR XIC B3:10/5 MOV N7:99 O:1.1 EOR
%   O:1.1  TOP_CONV_SPED %
% Rung: 5 %
SOR MOV N101:14 O:0.4 EOR
%   N101:14  FEED_WHL_SPD_SET  "feed wheel speed setting from hmi" %
%   O:0.4  FEED_WHEEL_SPED %
% Rung: 6 %
SOR XIO B3:4/10 XIC B3:3/0 MOV N7:20 O:0.4 EOR
%   B3:4/10  FEED_WHEEL_EN  "feed wheel run" %
%   B3:3/0  "bypass" %
%   O:0.4  FEED_WHEEL_SPED %
% Rung: 7 %
% bolt feeder speed %
SOR MOV N101:13 N7:26 EOR
%   N101:13  FEED_BOWL_SET_SPD %

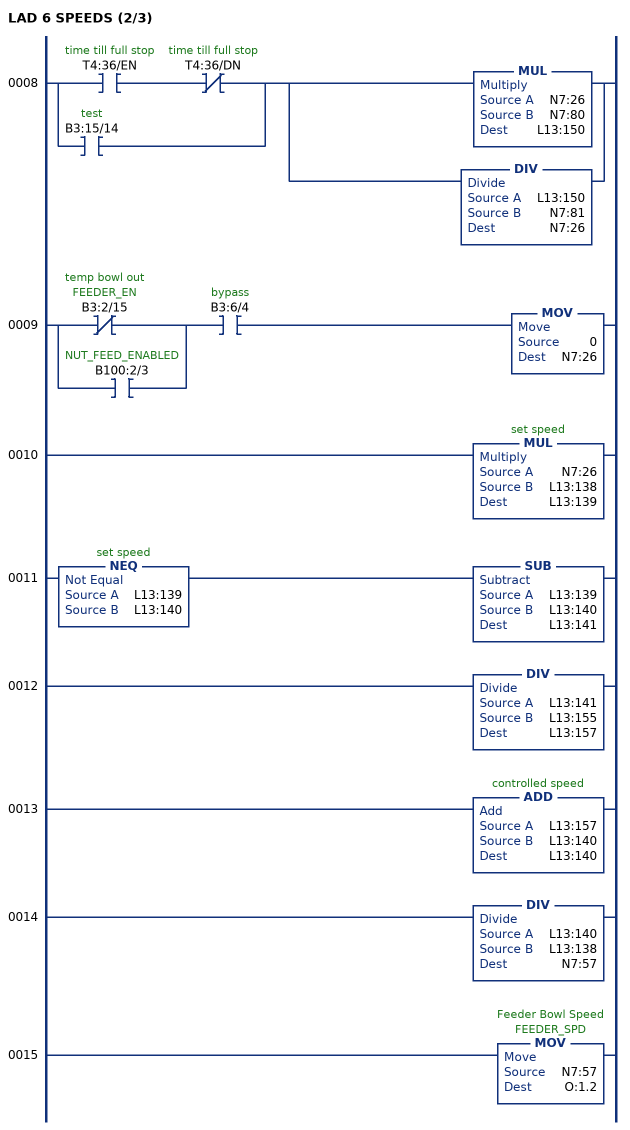
% Rung: 8 %
SOR BST XIC T4:36/EN XIO T4:36/DN NXB XIC B3:15/14 BND BST MUL N7:26 N7:80 L13:150 NXB DIV L13:150 N7:81 N7:26 BND EOR
%   T4:36  "time till full stop" %
%   B3:15/14  "test" %
% Rung: 9 %
SOR BST XIO B3:2/15 NXB XIC B100:2/3 BND XIC B3:6/4 MOV 0 N7:26 EOR
%   B3:2/15  FEEDER_EN  "temp bowl out" %
%   B100:2/3  NUT_FEED_ENABLED %
%   B3:6/4  "bypass" %
% Rung: 10 %
SOR MUL N7:26 L13:138 L13:139 EOR
%   L13:139  "set speed" %
% Rung: 11 %
SOR NEQ L13:139 L13:140 SUB L13:139 L13:140 L13:141 EOR
%   L13:139  "set speed" %
%   L13:140  "controlled speed" %
% Rung: 12 %
SOR DIV L13:141 L13:155 L13:157 EOR
% Rung: 13 %
SOR ADD L13:157 L13:140 L13:140 EOR
%   L13:140  "controlled speed" %
% Rung: 14 %
SOR DIV L13:140 L13:138 N7:57 EOR
%   L13:140  "controlled speed" %
% Rung: 15 %
SOR MOV N7:57 O:1.2 EOR
%   O:1.2  FEEDER_SPD  "Feeder Bowl Speed" %

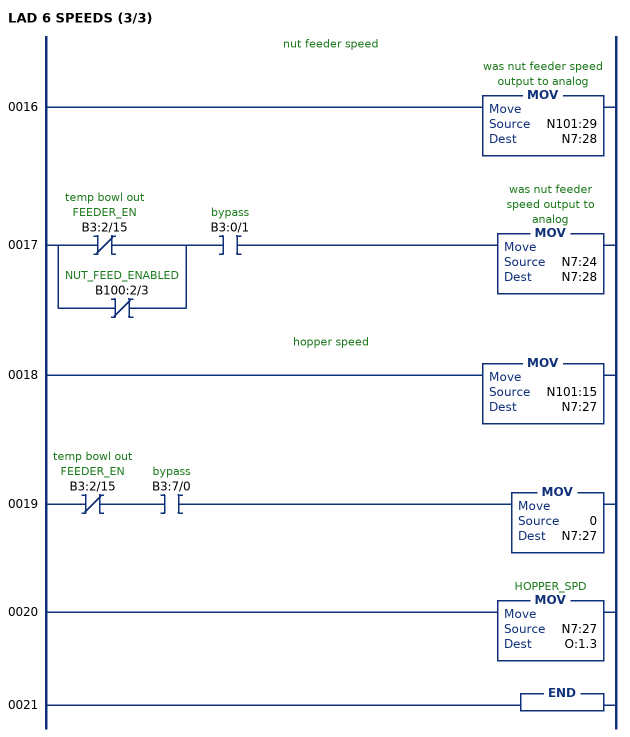
% Rung: 16 %
% nut feeder speed %
SOR MOV N101:29 N7:28 EOR
%   N101:29  "was nut feeder speed setting from hmi" %
%   N7:28  "was nut feeder speed output to analog" %
% Rung: 17 %
SOR BST XIO B3:2/15 NXB XIO B100:2/3 BND XIC B3:0/1 MOV N7:24 N7:28 EOR
%   B3:2/15  FEEDER_EN  "temp bowl out" %
%   B100:2/3  NUT_FEED_ENABLED %
%   B3:0/1  "bypass" %
%   N7:28  "was nut feeder speed output to analog" %
% Rung: 18 %
% hopper speed %
SOR MOV N101:15 N7:27 EOR
%   N101:15  HOPPER_SPD_SETTING  "hopper speed setting from hmi" %
% Rung: 19 %
SOR XIO B3:2/15 XIC B3:7/0 MOV 0 N7:27 EOR
%   B3:2/15  FEEDER_EN  "temp bowl out" %
%   B3:7/0  "bypass" %
% Rung: 20 %
SOR MOV N7:27 O:1.3 EOR
%   O:1.3  HOPPER_SPD %
% Rung: 21 %
SOR END EOR

LADDER 7 "HSC BOT"
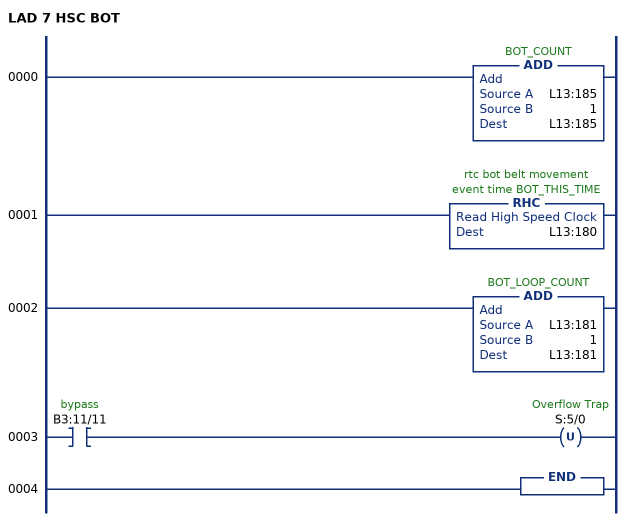
% Rung: 0 %
SOR ADD L13:185 1 L13:185 EOR
%   L13:185  BOT_COUNT %
% Rung: 1 %
SOR RHC L13:180 EOR
%   L13:180  BOT_THIS_TIME  "rtc bot belt movement event time" %
% Rung: 2 %
SOR ADD L13:181 1 L13:181 EOR
%   L13:181  BOT_LOOP_COUNT %
% Rung: 3 %
SOR XIC B3:11/11 OTU S:5/0 EOR
%   B3:11/11  "bypass" %
%   S:5/0  "Overflow Trap" %
% Rung: 4 %
SOR END EOR

LADDER 8 "HSC TOP"
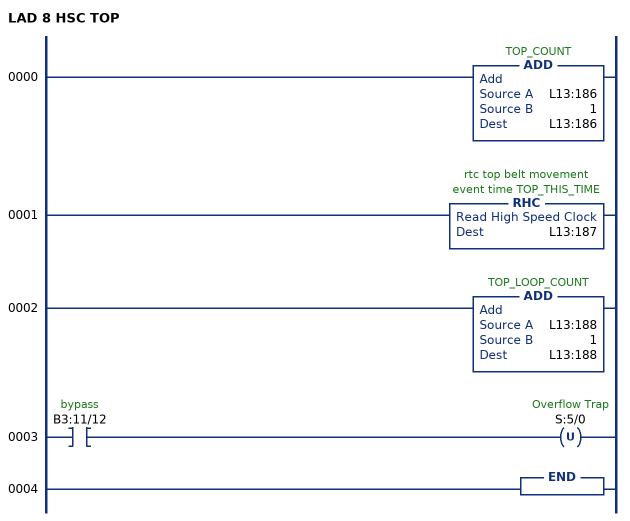
% Rung: 0 %
SOR ADD L13:186 1 L13:186 EOR
%   L13:186  TOP_COUNT %
% Rung: 1 %
SOR RHC L13:187 EOR
%   L13:187  TOP_THIS_TIME  "rtc top belt movement event time" %
% Rung: 2 %
SOR ADD L13:188 1 L13:188 EOR
%   L13:188  TOP_LOOP_COUNT %
% Rung: 3 %
SOR XIC B3:11/12 OTU S:5/0 EOR
%   B3:11/12  "bypass" %
%   S:5/0  "Overflow Trap" %
% Rung: 4 %
SOR END EOR

LADDER 9 "1 MS STI"    % high speed %
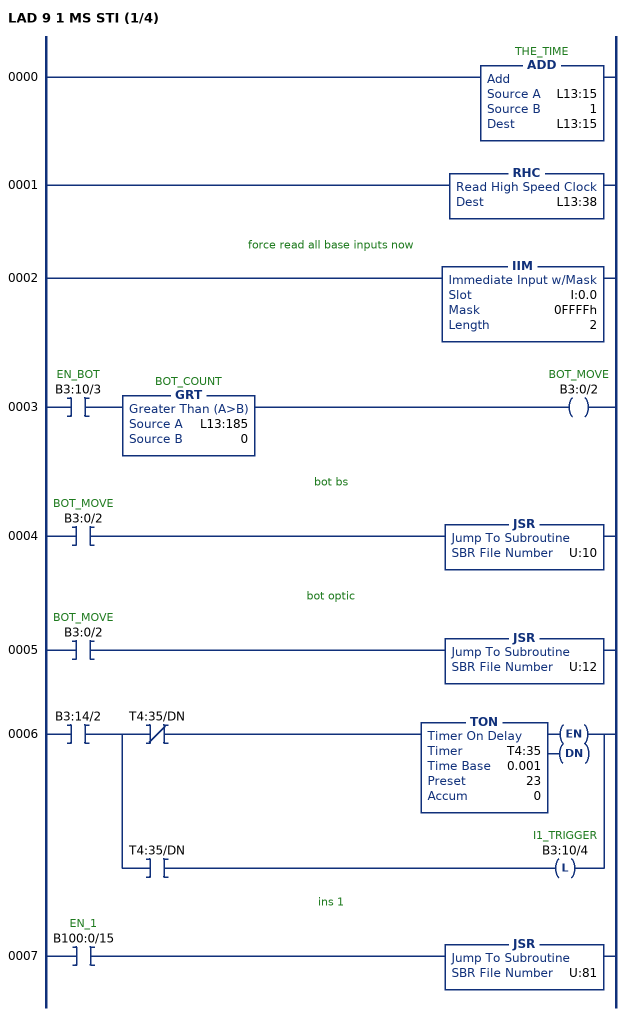
% Rung: 0 %
SOR ADD L13:15 1 L13:15 EOR
%   L13:15  THE_TIME %
% Rung: 1 %
SOR RHC L13:38 EOR
% Rung: 2 %
% force read all base inputs now %
SOR IIM I:0.0 0FFFFh 2 EOR
% Rung: 3 %
SOR XIC B3:10/3 GRT L13:185 0 OTE B3:0/2 EOR
%   B3:10/3  EN_BOT %
%   L13:185  BOT_COUNT %
%   B3:0/2  BOT_MOVE %
% Rung: 4 %
% bot bs %
SOR XIC B3:0/2 JSR U:10 EOR
%   B3:0/2  BOT_MOVE %
% Rung: 5 %
% bot optic %
SOR XIC B3:0/2 JSR U:12 EOR
%   B3:0/2  BOT_MOVE %
% Rung: 6 %
SOR XIC B3:14/2 BST XIO T4:35/DN TON T4:35 0.001 23 0 NXB XIC T4:35/DN OTL B3:10/4 BND EOR
%   B3:10/4  I1_TRIGGER %
% Rung: 7 %
% ins 1 %
SOR XIC B100:0/15 JSR U:81 EOR
%   B100:0/15  EN_1 %

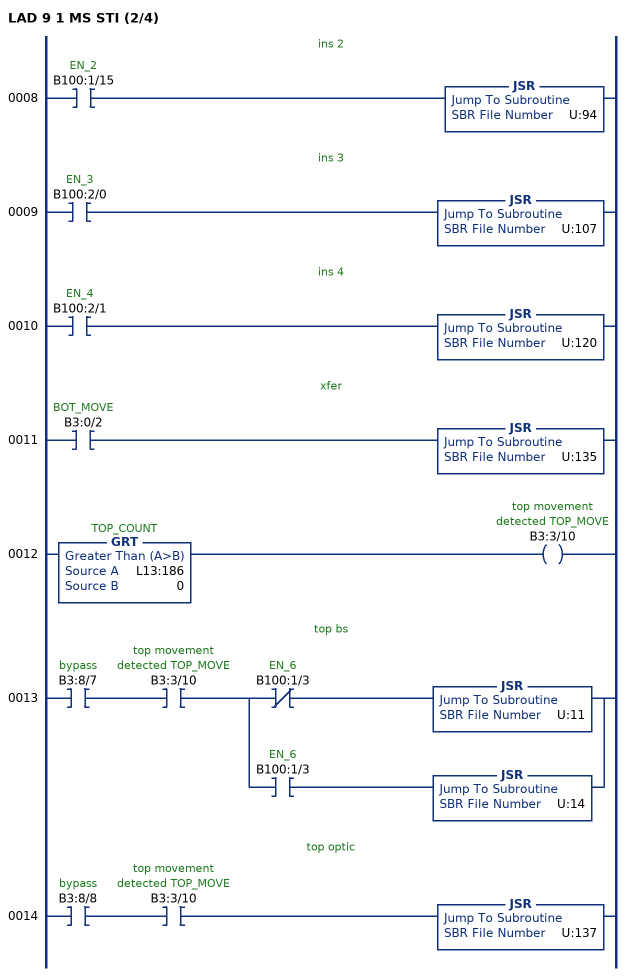
% Rung: 8 %
% ins 2 %
SOR XIC B100:1/15 JSR U:94 EOR
%   B100:1/15  EN_2 %
% Rung: 9 %
% ins 3 %
SOR XIC B100:2/0 JSR U:107 EOR
%   B100:2/0  EN_3 %
% Rung: 10 %
% ins 4 %
SOR XIC B100:2/1 JSR U:120 EOR
%   B100:2/1  EN_4 %
% Rung: 11 %
% xfer %
SOR XIC B3:0/2 JSR U:135 EOR
%   B3:0/2  BOT_MOVE %
% Rung: 12 %
SOR GRT L13:186 0 OTE B3:3/10 EOR
%   L13:186  TOP_COUNT %
%   B3:3/10  TOP_MOVE  "top movement detected" %
% Rung: 13 %
% top bs %
SOR XIC B3:8/7 XIC B3:3/10 BST XIO B100:1/3 JSR U:11 NXB XIC B100:1/3 JSR U:14 BND EOR
%   B3:8/7  "bypass" %
%   B3:3/10  TOP_MOVE  "top movement detected" %
%   B100:1/3  EN_6 %
% Rung: 14 %
% top optic %
SOR XIC B3:8/8 XIC B3:3/10 JSR U:137 EOR
%   B3:8/8  "bypass" %
%   B3:3/10  TOP_MOVE  "top movement detected" %

